FUNCTION_BLOCK FB_Coordinador_SFC

VAR_INPUT
    SFCPause: BOOL;
    SFCReset: BOOL;
    
    // Indicadores de sincronizacion
    Benido: BOOL := TRUE;
    Ejecuta: BOOL;
    
    // Indicadores de control
    Resume: BOOL;
    StepByStep: BOOL;
    
    // Parametros de sincronizacion
    PaleSituado: BOOL;
    Alimentado: BOOL;
    Cargado: BOOL;
    Girado: BOOL;
    Medido: BOOL;
    Rechazada: BOOL;
    Descargada: BOOL;
    Transferido: BOOL;
    
    
    // Parametros
    CondicionInicial: BOOL;
    UnidadesSolicitadas: UINT;
    
    Tapas : ARRAY[0..7] OF ST_POSICION;
    //TapaAuxRot : ST_POSICION; 
    //CLK: FB_Clock;
    
    TapaDeseada : ST_TAPA;
    //NumPiezasDes: UINT;
    cont: UINT;
    
END_VAR

VAR_OUTPUT
    Acabhe: BOOL;
    ListoKalisto: BOOL;
    
    // Parametros de sincronizacion
    SituaPale: BOOL;
    Alimenta: BOOL;
    Carga: BOOL;
    Gira: BOOL;
    Mide: BOOL;
    Descarga: BOOL;
    Rechaza: BOOL;
    Transfiere : BOOL;
    
    
    // Salidas
     LamparaAlarma: BOOL;
    LamparaMarcha: BOOL;
END_VAR
   
VAR_IN_OUT
   
END_VAR

VAR
     // Bloques funcionales
    CLK: FB_Clock;
    Deseada : BOOL;
    Eliminada : BOOL; 
END_VAR

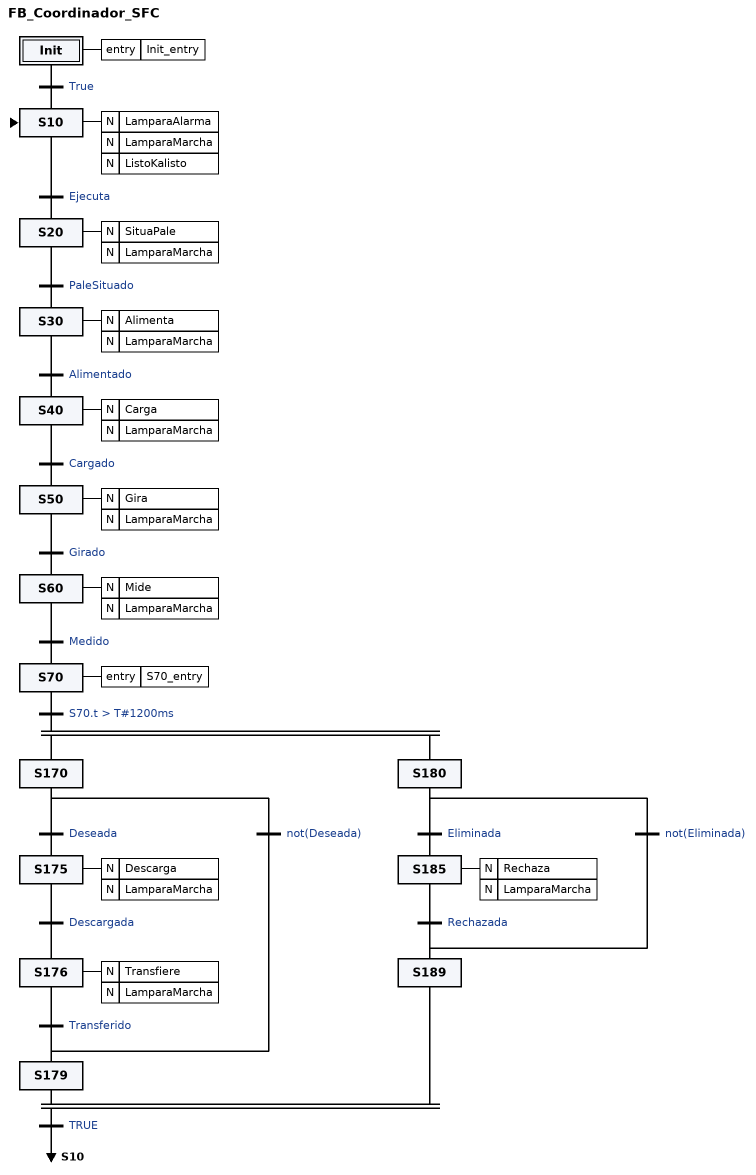
INITIAL_STEP Init:
    Init_entry(P1);  // entry action
END_STEP
TRANSITION FROM Init TO S10
    := True;
END_TRANSITION
STEP S10:
    LamparaAlarma(N);
    LamparaMarcha(N);
    ListoKalisto(N);
END_STEP
TRANSITION FROM S10 TO S20
    := Ejecuta;
END_TRANSITION
STEP S20:
    SituaPale(N);
    LamparaMarcha(N);
END_STEP
TRANSITION FROM S20 TO S30
    := PaleSituado;
END_TRANSITION
STEP S30:
    Alimenta(N);
    LamparaMarcha(N);
END_STEP
TRANSITION FROM S30 TO S40
    := Alimentado;
END_TRANSITION
STEP S40:
    Carga(N);
    LamparaMarcha(N);
END_STEP
TRANSITION FROM S40 TO S50
    := Cargado;
END_TRANSITION
STEP S50:
    Gira(N);
    LamparaMarcha(N);
END_STEP
TRANSITION FROM S50 TO S60
    := Girado;
END_TRANSITION
STEP S60:
    Mide(N);
    LamparaMarcha(N);
END_STEP
TRANSITION FROM S60 TO S70
    := Medido;
END_TRANSITION
STEP S70:
    S70_entry(P1);  // entry action
END_STEP
TRANSITION FROM S70 TO (S170, S180)
    := S70.t > T#1200ms;
END_TRANSITION
STEP S170:
END_STEP
TRANSITION FROM S170 TO S175
    := Deseada;
END_TRANSITION
STEP S175:
    Descarga(N);
    LamparaMarcha(N);
END_STEP
TRANSITION FROM S175 TO S176
    := Descargada;
END_TRANSITION
STEP S176:
    Transfiere(N);
    LamparaMarcha(N);
END_STEP
TRANSITION FROM S176 TO S179
    := Transferido;
END_TRANSITION
TRANSITION FROM S170 TO S179
    := not(Deseada);
END_TRANSITION
STEP S179:
END_STEP
STEP S180:
END_STEP
TRANSITION FROM S180 TO S185
    := Eliminada;
END_TRANSITION
STEP S185:
    Rechaza(N);
    LamparaMarcha(N);
END_STEP
TRANSITION FROM S185 TO S189
    := Rechazada;
END_TRANSITION
TRANSITION FROM S180 TO S189
    := not(Eliminada);
END_TRANSITION
STEP S189:
END_STEP
TRANSITION FROM (S179, S189) TO S10
    := TRUE;
END_TRANSITION

ACTION Init_entry:

Tapas[0].Ocupada := 0;
Tapas[1].Ocupada := 0;
Tapas[2].Ocupada := 0;
Tapas[3].Ocupada := 0;
Tapas[4].Ocupada := 0;
Tapas[5].Ocupada := 0;
Tapas[6].Ocupada := 0;
Tapas[7].Ocupada := 0;
END_ACTION

ACTION S10_exit:

END_ACTION

ACTION S70_entry:
Deseada := (Tapas[7].Ocupada AND Tapas[7].Tapa.Alta = TapaDeseada.Alta AND Tapas[7].Tapa.Clara = TapaDeseada.Clara AND Tapas[7].Tapa.Metalica = TapaDeseada.Metalica);

Eliminada := (Tapas[6].Ocupada AND NOT(Tapas[6].Tapa.Alta = TapaDeseada.Alta AND Tapas[6].Tapa.Clara = TapaDeseada.Clara AND Tapas[6].Tapa.Metalica = TapaDeseada.Metalica));
END_ACTION

END_FUNCTION_BLOCK

(* stored: Version 1.1.0.1, ProductVersion 3.1.4024.12
   POU FB_Coordinador_SFC: Id {8281f6e9-331f-40c9-b896-41f2f2d0b403}, SpecialFunc None
   Action Init_entry: Id {b24d784b-b2a2-4993-8844-fd421696650b}
   Action S10_exit: Id {dfc64b29-8306-4ec4-a33d-02f6403a530f}
   Action S70_entry: Id {7c93b1b9-da26-4bbc-b082-365743a32e80} *)
